PROGRAM MAIN
VAR
	counter : REAL := 1;
	toggle: BOOL;
	pushButton	:BOOL;
	clickButton :BOOL;
	light 		:BOOL;
	t1 			:TON;
	tr1			:R_TRIG;
	pulse		:TP;
	
	sine		:REAL;
END_VAR

prgPumpControl();
IF counter > 4000 THEN
	counter := 0;
ELSE
	counter := counter+1;
END_IF

sine := SIN(counter/500);




//counter:= counter+2;

//t1(IN:=pushButton, PT:= T#5S, Q=> light, ET=> );
//t1(PT:= T#5S );
//t1.IN:=pushButton;

//pulse(IN:= pushButton, PT:= T#500MS, Q=> , ET=> ); 
//tr1(CLK:= clickButton, Q=> light);

//IF counter > 1000 THEN
//	counter := 0;
//	toggle := NOT toggle;
	
//	NEWSUBROUTINE(input:=toggle);
//	//comment
//	(*
//	multi
//	line 
//	comment
//	*)
//END_IF

ACTION ACT:
// NETWORK 1
END_ACTION

END_PROGRAM

(* stored: Version 1.1.0.1, ProductVersion 3.1.4024.13
   POU MAIN: Id {c64330fb-d57a-4062-809d-d9c7753c4dc9}, SpecialFunc None
   Action ACT: Id {5b52bf2f-4d04-42d6-84de-942ff01eddc7} *)
